{attribute 'linkalways'} 
{attribute 'no_explicit_call' := 'This FB is a CLASS and must be accessed using methods or properties'}
{attribute 'enable_dynamic_creation'}
FUNCTION_BLOCK FINAL LN_LREAL EXTENDS Node
VAR
	in : _LREAL(0.0);
	out : _LREAL(0.0);
END_VAR

METHOD PUBLIC Clone : I_Node
VAR
	pNode : POINTER TO LN_LREAL;
END_VAR
pNode := __NEW(LN_LREAL);
Clone := pNode^;
END_METHOD

METHOD FB_init : BOOL
VAR_INPUT
	bInitRetains : BOOL; // if TRUE, the retain variables are initialized (warm start / cold start)
	bInCopyCode : BOOL;  // if TRUE, the instance afterwards gets moved into the copy code (online change)
END_VAR
AddInput('in',THIS^.in);
AddOutput('out', THIS^.out);
END_METHOD

METHOD PROTECTED OnExecute
VAR
END_VAR
out.Value := LN(in.Value);
END_METHOD

END_FUNCTION_BLOCK

(* stored: Version 1.1.0.1, ProductVersion 3.1.4024.15
   POU LN_LREAL: Id {1734fa61-d5e3-41a5-84ef-79a0cea53491}, SpecialFunc None
   Folder Constructor: Id {9eb4bba5-40eb-490a-aea0-5f3c39d742b2}
   Method Clone: Id {83186980-4416-4a7d-a2e2-8b425978944e}
   Method FB_init: Id {db7cccf3-d31b-45b1-81db-7ddf67ff1ea5}
   Method OnExecute: Id {cf4cb419-7763-4873-9cf3-aeb6d250b974} *)
